(* This function is the equivalent of FREQ_MEASURE from codesys's utility library.
   It emulates their wacky API that tries to auto-detect specific errors *)
FUNCTION_BLOCK FB_FreqMeasure
VAR_INPUT
	// Input signal
    IN: BOOL;
	// Number of periods to average the frequency over.
	// Must be between 1 and 100
    PERIODS: UINT := 1;
	// Reset all parameters to 0
    RESET: BOOL;
END_VAR
VAR_OUTPUT
	// Frequency in HZ
    OUT: REAL;
	// FALSE until we've measured at least PERIODS periods, or if distance between two rising edges is > 3 * OUT
    VALID: BOOL;
END_VAR
VAR
	RisingEnableEdge: R_TRIG;
	FallingEnableEdge : F_TRIG;
    STARTED: BOOL;
    RISETIME: TIME;
	AveragePeriod : FB_MovingAverageReal;
	// Difference in time between current and last rising edge
    DIFF: DINT;
	// Array of time differences for each period
    TIMEDIFF: ARRAY[0..99] OF LREAL;
	// How many periods we have counted so far
    COUNT: UINT;
	SYSTIMEMS : TIME;          
END_VAR
VAR_TEMP
	OutTemp : LREAL;
END_VAR


IF Reset THEN
    VALID := FALSE;
    COUNT := 0;
    STARTED := FALSE;
    OUT := 0;
    RETURN;
END_IF

RisingEnableEdge(CLK := IN);
FallingEnableEdge(CLK := IN);

(* We care only about whether we are the beginning or the end of the signal.
   If we are at the beginning, we store the current time the signal rose.
   If we are the end, we look at the current time, subtract the rise time,
   and add the signal time period to the period array.
   Once we have collected the requested number of periods, we start averaging
   and mark ourselves valid. *)
IF RisingEnableEdge.Q OR FallingEnableEdge.Q THEN
	// The tming mechanism depends on the PLC. What we expect is something that produces milliseconds.
	// The only requirement is that the difference between the two times represent the signal period in millliseconds
	SYSTIMEMS := ULINT_TO_TIME(F_GetTaskTime() / TC2_Utilities.SYSTEMTIME_TICKSPERMSEC64);
    IF FallingEnableEdge.Q AND STARTED THEN
		DIFF := TIME_TO_DINT(SYSTIMEMS - RISETIME);
		// We assume time never goes backwards for real. Unfortunately, the API of this call does
		// not give us a way to express errors easily.
        IF Diff > 0 THEN
			// Emulate the weird behavior of CODESYS FREQ_MEASURE
			IF VALID AND Diff > 3000 * REAL_TO_DINT(OUT) THEN
				VALID := FALSE;
				COUNT := 0;
				RETURN;
			END_IF
			// Compute moving average over periods
			AveragePeriod(ValueToAdd := DINT_TO_REAL(DIFF),
						  AverageArray := TIMEDIFF,
						  NumValuesToUse := PERIODS,
						  CurrentValue => OutTemp);
			Out := LREAL_TO_REAL (OutTemp); 
            COUNT := MIN(COUNT + 1, PERIODS);
			// Go valid once we have the minimum number of periods to average over.
            VALID := COUNT = PERIODS;
        END_IF
		STARTED := FALSE;
		RETURN;
    END_IF
    STARTED := TRUE;
    RISETIME := SYSTIMEMS;
END_IF

END_FUNCTION_BLOCK

(* stored: Version 1.1.0.1, ProductVersion 3.1.4022.16
   POU FB_FreqMeasure: Id {3d6d3d65-e18a-4fc3-a773-f23be8247d43}, SpecialFunc None *)
